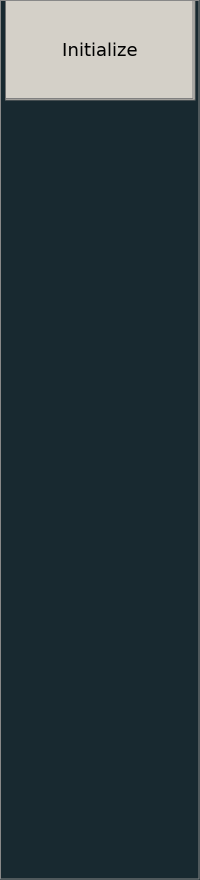
VISUALIZATION NavBarUninitialized_1  // 200x880
VAR_IN_OUT
	btnInitialize	: BOOL;	(*  *)
END_VAR
    Button (5,0 190x100), "Initialize"
        tap btnInitialize
END_VISUALIZATION

(* stored: Version 1.1.0.1, ProductVersion 3.1.4024.12
   Visu NavBarUninitialized_1: Id {8e7b723a-1467-46dc-ba98-f3092ffa802b} *)
